TYPE ST_System_BHKW_Zustand :
STRUCT
	Betrieb_Anford				: BOOL;
	Betrieb_Soll				: BOOL;
	Betrieb						: BOOL;
	Betrieb_ohne_Komm			: BOOL;

	Regelung_Sollw				: REAL;

	Netze_Anford				: ST_Zustand_Netze_Anford;

	Netz_HW_Anford				: ST_Zustand_Netz_Anford;

	Freigabe					: BOOL;
	Freigabe_Deakt				: BOOL;
	Freigabe_Code				: WORD;

	Stoerung					: BOOL;
	Stoerung_Code				: WORD;

	Warnung						: BOOL;
	Warnung_Code				: WORD;

	Status						: SINT;
	Status_Vorl_Stellventil		: BOOL;
	Status_Vorl_Pumpe			: BOOL;
	Status_Vorl_BHKW			: BOOL;
	Status_Nachl_Stellventil	: BOOL;
	Status_Nachl_Pumpe			: BOOL;
	Status_Nachl_BHKW			: BOOL;
	Status_Nachl_BHKW_ohne_Komm	: BOOL;
	Status_BHKW_ueberhitzt		: BOOL;

	Quittierung					: BOOL;

END_STRUCT
END_TYPE

(* stored: Version 1.1.0.1, ProductVersion 3.1.4024.9
   DUT ST_System_BHKW_Zustand: Id {b735e499-0cd8-492f-a2e2-26f5d8113fae} *)
